TEXTLIST LineLoadClose
  0 = 'LineLoad_None'
  1 = 'Line0LoadClose'
  2 = 'Line1LoadClose'
   = ''
END_TEXTLIST

(* stored: Version 1.1.0.1, ProductVersion 3.1.4024.3
   TextList LineLoadClose: Id {d63b00bf-042e-4bad-b7d3-7741a0326ed6} *)
